(* CODESYS project addition_1.xml

Project tree, tasks and I/O mapping:
  function addition_1 [ST]
*)

// addition_1
FUNCTION addition_1 : STRING
VAR_INPUT
END_VAR
VAR
END_VAR

addition_1		:=		FU_sConcat3(s1:='1',s2:='2',s3:='3');

END_FUNCTION
